PROGRAM ManualCtrl
VAR

	Manual1PageEnable: BOOL;
	Manual2PageEnable: BOOL;
	MPAGE1: MANUAL_PAGE;
	MPAGE2: MANUAL_PAGE;

END_VAR

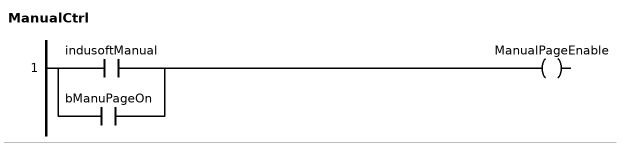
// NETWORK 1
ManualPageEnable := indusoftManual OR bManuPageOn;

END_PROGRAM

(* stored: Version 1.1.0.1, ProductVersion 3.1.4024.12
   POU ManualCtrl: Id {54ad4890-b44d-4d25-b03a-039575ab40c7}, SpecialFunc None *)
